    Win32ErrorCodes.ERROR_IPSEC_IKE_NO_POLICY:
        Win32ErrorCodeDescription := 'No policy configured.';
    Win32ErrorCodes.ERROR_IPSEC_IKE_INVALID_SIGNATURE:
        Win32ErrorCodeDescription := 'Failed to verify signature.';
    Win32ErrorCodes.ERROR_IPSEC_IKE_KERBEROS_ERROR:
        Win32ErrorCodeDescription := 'Failed to authenticate using Kerberos.';
    Win32ErrorCodes.ERROR_IPSEC_IKE_NO_PUBLIC_KEY:
        Win32ErrorCodeDescription := 'Peers certificate did not have a public key.';
    Win32ErrorCodes.ERROR_IPSEC_IKE_PROCESS_ERR:
        Win32ErrorCodeDescription := 'Error processing error payload.';
    Win32ErrorCodes.ERROR_IPSEC_IKE_PROCESS_ERR_SA:
        Win32ErrorCodeDescription := 'Error processing SA payload.';
    Win32ErrorCodes.ERROR_IPSEC_IKE_PROCESS_ERR_PROP:
        Win32ErrorCodeDescription := 'Error processing Proposal payload.';
    Win32ErrorCodes.ERROR_IPSEC_IKE_PROCESS_ERR_TRANS:
        Win32ErrorCodeDescription := 'Error processing Transform payload.';
    Win32ErrorCodes.ERROR_IPSEC_IKE_PROCESS_ERR_KE:
        Win32ErrorCodeDescription := 'Error processing KE payload.';
    Win32ErrorCodes.ERROR_IPSEC_IKE_PROCESS_ERR_ID:
        Win32ErrorCodeDescription := 'Error processing ID payload.';
    Win32ErrorCodes.ERROR_IPSEC_IKE_PROCESS_ERR_CERT:
        Win32ErrorCodeDescription := 'Error processing Cert payload.';
    Win32ErrorCodes.ERROR_IPSEC_IKE_PROCESS_ERR_CERT_REQ:
        Win32ErrorCodeDescription := 'Error processing Certificate Request payload.';
    Win32ErrorCodes.ERROR_IPSEC_IKE_PROCESS_ERR_HASH:
        Win32ErrorCodeDescription := 'Error processing Hash payload.';
    Win32ErrorCodes.ERROR_IPSEC_IKE_PROCESS_ERR_SIG:
        Win32ErrorCodeDescription := 'Error processing Signature payload.';
    Win32ErrorCodes.ERROR_IPSEC_IKE_PROCESS_ERR_NONCE:
        Win32ErrorCodeDescription := 'Error processing Nonce payload.';
    Win32ErrorCodes.ERROR_IPSEC_IKE_PROCESS_ERR_NOTIFY:
        Win32ErrorCodeDescription := 'Error processing Notify payload.';
    Win32ErrorCodes.ERROR_IPSEC_IKE_PROCESS_ERR_DELETE:
        Win32ErrorCodeDescription := 'Error processing Delete Payload.';
    Win32ErrorCodes.ERROR_IPSEC_IKE_PROCESS_ERR_VENDOR:
        Win32ErrorCodeDescription := 'Error processing VendorId payload.';
    Win32ErrorCodes.ERROR_IPSEC_IKE_INVALID_PAYLOAD:
        Win32ErrorCodeDescription := 'Invalid payload received.';
    Win32ErrorCodes.ERROR_IPSEC_IKE_LOAD_SOFT_SA:
        Win32ErrorCodeDescription := 'Soft SA loaded.';
    Win32ErrorCodes.ERROR_IPSEC_IKE_SOFT_SA_TORN_DOWN:
        Win32ErrorCodeDescription := 'Soft SA torn down.';
    Win32ErrorCodes.ERROR_IPSEC_IKE_INVALID_COOKIE:
        Win32ErrorCodeDescription := 'Invalid cookie received..';
    Win32ErrorCodes.ERROR_IPSEC_IKE_NO_PEER_CERT:
        Win32ErrorCodeDescription := 'Peer failed to send valid machine certificate.';
    Win32ErrorCodes.ERROR_IPSEC_IKE_PEER_CRL_FAILED:
        Win32ErrorCodeDescription := 'Certification Revocation check of peers certificate failed.';
    Win32ErrorCodes.ERROR_IPSEC_IKE_POLICY_CHANGE:
        Win32ErrorCodeDescription := 'New policy invalidated SAs formed with old policy.';
    Win32ErrorCodes.ERROR_IPSEC_IKE_NO_MM_POLICY:
        Win32ErrorCodeDescription := 'There is no available Main Mode IKE policy.';
    Win32ErrorCodes.ERROR_IPSEC_IKE_NOTCBPRIV:
        Win32ErrorCodeDescription := 'Failed to enabled TCB privilege.';
    Win32ErrorCodes.ERROR_IPSEC_IKE_SECLOADFAIL:
        Win32ErrorCodeDescription := 'Failed to load SECURITY.DLL.';
    Win32ErrorCodes.ERROR_IPSEC_IKE_FAILSSPINIT:
        Win32ErrorCodeDescription :=
            'Failed to obtain security function table dispatch address from SSPI.';
    Win32ErrorCodes.ERROR_IPSEC_IKE_FAILQUERYSSP:
        Win32ErrorCodeDescription := 'Failed to query Kerberos package to obtain max token size.';
    Win32ErrorCodes.ERROR_IPSEC_IKE_SRVACQFAIL:
        Win32ErrorCodeDescription := 'Failed to obtain Kerberos server credentials for ISAKMP/ERROR_IPSEC_IKE service. Kerberos authentication will not function. The most likely reason for this is lack of domain membership. This is normal if your computer is a member of a workgroup.';
    Win32ErrorCodes.ERROR_IPSEC_IKE_SRVQUERYCRED:
        Win32ErrorCodeDescription := 'Failed to determine SSPI principal name for ISAKMP/ERROR_IPSEC_IKE service (QueryCredentialsAttributes).';
    Win32ErrorCodes.ERROR_IPSEC_IKE_GETSPIFAIL:
        Win32ErrorCodeDescription := 'Failed to obtain new SPI for the inbound SA from Ipsec driver. The most common cause for this is that the driver does not have the correct filter. Check your policy to verify the filters.';
    Win32ErrorCodes.ERROR_IPSEC_IKE_INVALID_FILTER:
        Win32ErrorCodeDescription := 'Given filter is invalid.';
    Win32ErrorCodes.ERROR_IPSEC_IKE_OUT_OF_MEMORY:
        Win32ErrorCodeDescription := 'Memory allocation failed.';
    Win32ErrorCodes.ERROR_IPSEC_IKE_ADD_UPDATE_KEY_FAILED:
        Win32ErrorCodeDescription := 'Failed to add Security Association to IPSec Driver. The most common cause for this is if the IKE negotiation took too long to complete. If the problem persists, reduce the load on the faulting machine.';
    Win32ErrorCodes.ERROR_IPSEC_IKE_INVALID_POLICY:
        Win32ErrorCodeDescription := 'Invalid policy.';
    Win32ErrorCodes.ERROR_IPSEC_IKE_UNKNOWN_DOI:
        Win32ErrorCodeDescription := 'Invalid DOI.';
    Win32ErrorCodes.ERROR_IPSEC_IKE_INVALID_SITUATION:
        Win32ErrorCodeDescription := 'Invalid situation.';
    Win32ErrorCodes.ERROR_IPSEC_IKE_DH_FAILURE:
        Win32ErrorCodeDescription := 'Diffie-Hellman failure.';
    Win32ErrorCodes.ERROR_IPSEC_IKE_INVALID_GROUP:
        Win32ErrorCodeDescription := 'Invalid Diffie-Hellman group.';
    Win32ErrorCodes.ERROR_IPSEC_IKE_ENCRYPT:
        Win32ErrorCodeDescription := 'Error encrypting payload.';
    Win32ErrorCodes.ERROR_IPSEC_IKE_DECRYPT:
        Win32ErrorCodeDescription := 'Error decrypting payload.';
    Win32ErrorCodes.ERROR_IPSEC_IKE_POLICY_MATCH:
        Win32ErrorCodeDescription := 'Policy match error.';
    Win32ErrorCodes.ERROR_IPSEC_IKE_UNSUPPORTED_ID:
        Win32ErrorCodeDescription := 'Unsupported ID.';
    Win32ErrorCodes.ERROR_IPSEC_IKE_INVALID_HASH:
        Win32ErrorCodeDescription := 'Hash verification failed.';
    Win32ErrorCodes.ERROR_IPSEC_IKE_INVALID_HASH_ALG:
        Win32ErrorCodeDescription := 'Invalid hash algorithm.';
    Win32ErrorCodes.ERROR_IPSEC_IKE_INVALID_HASH_SIZE:
        Win32ErrorCodeDescription := 'Invalid hash size.';
    Win32ErrorCodes.ERROR_IPSEC_IKE_INVALID_ENCRYPT_ALG:
        Win32ErrorCodeDescription := 'Invalid encryption algorithm.';
    Win32ErrorCodes.ERROR_IPSEC_IKE_INVALID_AUTH_ALG:
        Win32ErrorCodeDescription := 'Invalid authentication algorithm.';
    Win32ErrorCodes.ERROR_IPSEC_IKE_INVALID_SIG:
        Win32ErrorCodeDescription := 'Invalid certificate signature.';
    Win32ErrorCodes.ERROR_IPSEC_IKE_LOAD_FAILED:
        Win32ErrorCodeDescription := 'Load failed.';
    Win32ErrorCodes.ERROR_IPSEC_IKE_RPC_DELETE:
        Win32ErrorCodeDescription := 'Deleted via RPC call.';
    Win32ErrorCodes.ERROR_IPSEC_IKE_BENIGN_REINIT:
        Win32ErrorCodeDescription :=
            'Temporary state created to perform reinitialization. This is not a real failure.';
    Win32ErrorCodes.ERROR_IPSEC_IKE_INVALID_RESPONDER_LIFETIME_NOTIFY:
        Win32ErrorCodeDescription := 'The lifetime value received in the Responder Lifetime Notify is below the Windows 2000 configured minimum value. Please fix the policy on the peer machine.';
    Win32ErrorCodes.ERROR_IPSEC_IKE_QM_LIMIT_REAP:
        Win32ErrorCodeDescription := 'SA reaped because QM limit was reached.';
    Win32ErrorCodes.ERROR_IPSEC_IKE_INVALID_CERT_KEYLEN:
        Win32ErrorCodeDescription :=
            'Key length in certificate is too small for configured security requirements.';
    Win32ErrorCodes.ERROR_IPSEC_IKE_MM_LIMIT:
        Win32ErrorCodeDescription := 'Max number of established MM SAs to peer exceeded.';
    Win32ErrorCodes.ERROR_IPSEC_IKE_NEGOTIATION_DISABLED:
        Win32ErrorCodeDescription := 'IKE received a policy that disables negotiation.';
    Win32ErrorCodes.ERROR_IPSEC_IKE_QM_LIMIT:
        Win32ErrorCodeDescription :=
            'Reached maximum quick mode limit for the main mode. New main mode will be started.';
ELSE
    Win32ErrorCodeDescription := 'Unknown Win32 error code.';
END_CASE

END_FUNCTION

// ---- NC_Tests/ToNcErrorCode_Tests.TcPOU
FUNCTION_BLOCK ToNcErrorCode_Tests EXTENDS FB_TestSuite

ConversionOfValidErrorCode();
ConversionOfInvalidErrorCode();

METHOD ConversionOfInvalidErrorCode
TcUnit.TEST('ConversionOfInvalidErrorCode');

AssertEquals_DINT(
    Expected:=NcErrorCodes.ERR_UNKNOWN,
    Actual:=ToNcErrorCode(1234567),
    Message:='Error conversion not correct.'
);

TcUnit.TEST_FINISHED();
END_METHOD

METHOD ConversionOfValidErrorCode
TcUnit.TEST('ConversionOfValidErrorCode');

AssertEquals_UDINT(
    Expected:=NcErrorCodes.CONTROLLER_ERROR_DRIVE_ADDRESS,
    Actual:=ToNcErrorCode(17730),
    Message:='Error conversion not correct.'
);

TcUnit.TEST_FINISHED();
END_METHOD

END_FUNCTION_BLOCK

// ---- NC/ToNcErrorCode.TcPOU
(*
Convert a NC error code of type UDINT to the NcErrorCodes datatype.

## Example
```
ncErrorId := 17693;
ncErrorCode := ToNcErrorCode(ncErrorId); // CONTROLLER_ERROR_DEAD_RANGE_NOT_ALLOWED;
```

## Source
https://infosys.beckhoff.com/content/1033/tc3ncerrcode/1521556875.html?id=2911757239699425890
*)
FUNCTION ToNcErrorCode : NcErrorCodes
VAR_INPUT
    errorCode : UDINT;
END_VAR

CASE errorCode OF
    17664:
        ToNcErrorCode := NcErrorCodes.CONTROLLER_ERROR_CONTROLLER_ID_NOT_ALLOWED;
    17665:
        ToNcErrorCode := NcErrorCodes.CONTROLLER_ERROR_CONTROLLER_TYPE_NOT_ALLOWED;
    17666:
        ToNcErrorCode := NcErrorCodes.CONTROLLER_ERROR_OPERATION_MODE_CONTROLLER_NOT_ALLOWED;
    17667:
        ToNcErrorCode :=
            NcErrorCodes.CONTROLLER_ERROR_WEIGHTING_OF_THE_VELOCITY_PRE_CONTROL_NOT_ALLOWED;
    17668:
        ToNcErrorCode := NcErrorCodes.CONTROLLER_ERROR_LAG_ERROR_MONITOR_POSITION_NOT_ALLOWED;
    17669:
        ToNcErrorCode := NcErrorCodes.CONTROLLER_ERROR_LAG_MONITORING_VELOCITY_NOT_ALLOWED;
    17670:
        ToNcErrorCode := NcErrorCodes.CONTROLLER_ERROR_LAG_ERROR_WINDOW_POSITION_NOT_ALLOWED;
    17671:
        ToNcErrorCode := NcErrorCodes.CONTROLLER_ERROR_LAG_ERROR_FILTER_TIME_POSITION_NOT_ALLOWED;
    17672:
        ToNcErrorCode := NcErrorCodes.CONTROLLER_ERROR_LAG_ERROR_WINDOW_VELOCITY_NOT_ALLOWED;
    17673:
        ToNcErrorCode := NcErrorCodes.CONTROLLER_ERROR_LAG_ERROR_FILTER_TIME_VELOCITY_NOT_ALLOWED;
    17674:
        ToNcErrorCode := NcErrorCodes
            .CONTROLLER_ERROR_CONTROLLER_OUTPUT_LIMITATION_OUTPUT_LIMITATION_NOT_ALLOWED;
    17680:
        ToNcErrorCode :=
            NcErrorCodes.CONTROLLER_ERROR_PROPORTIONAL_GAIN_KV_OR_KP_CONTROLLER_NOT_ALLOWED;
    17681:
        ToNcErrorCode :=
            NcErrorCodes.CONTROLLER_ERROR_INTEGRAL_ACTION_TIME_TN_CONTROLLER_NOT_ALLOWED_POSITION;
    17682:
        ToNcErrorCode :=
            NcErrorCodes.CONTROLLER_ERROR_RATE_TIME_TV_CONTROLLER_NOT_ALLOWED_POSITION;
    17683:
        ToNcErrorCode :=
            NcErrorCodes.CONTROLLER_ERROR_DAMPING_TIME_TD_CONTROLLER_NOT_ALLOWED_POSITION;
    17684:
        ToNcErrorCode := NcErrorCodes
            .CONTROLLER_ERROR_ACTIVATION_OF_THE_AUTOMATIC_OFFSET_CALIBRATION_NOT_ALLOWED;
    17685:
        ToNcErrorCode := NcErrorCodes
            .CONTROLLER_ERROR_ADDITIONAL_PROPORTIONAL_GAIN_KV_OR_KP_CONTROLLER_NOT_ALLOWED;
    17686:
        ToNcErrorCode := NcErrorCodes
            .CONTROLLER_ERROR_REFERENCE_VELOCITY_FOR_ADDITIONAL_PROP_GAIN_CONTROLLER_NOT_ALLOWED;
    17687:
        ToNcErrorCode := NcErrorCodes.CONTROLLER_ERROR_PROPORTIONAL_GAIN_PA_PROPORTION_NOT_ALLOWED;
    17688:
        ToNcErrorCode := NcErrorCodes.CONTROLLER_ERROR_PROPORTIONAL_GAIN_KV_CONTROLLER_NOT_ALLOWED;
    17689:
        ToNcErrorCode :=
            NcErrorCodes.CONTROLLER_ERROR_INTEGRAL_ACTION_TIME_TN_CONTROLLER_NOT_ALLOWED_VELOCITY;
    17692:
        ToNcErrorCode := NcErrorCodes.CONTROLLER_ERROR_VELOCITY_FILTER_TIME_NOT_ALLOWED;
    17693:
        ToNcErrorCode := NcErrorCodes.CONTROLLER_ERROR_DEAD_RANGE_NOT_ALLOWED;
    17695:
        ToNcErrorCode := NcErrorCodes.CONTROLLER_ERROR_PROPORTIONAL_GAIN_KCP_NOT_ALLOWED;
    17696:
        ToNcErrorCode := NcErrorCodes.CONTROLLER_ERROR_RATE_TIME_TV_CONTROLLER_NOT_ALLOWED;
    17697:
        ToNcErrorCode := NcErrorCodes.CONTROLLER_ERROR_DAMPING_TIME_TD_CONTROLLER_NOT_ALLOWED;
    17698:
        ToNcErrorCode := NcErrorCodes.CONTROLLER_ERROR_LIMITATION_OF_THE_I_PART_NOT_ALLOWED;
    17699:
        ToNcErrorCode := NcErrorCodes.CONTROLLER_ERROR_LIMITATION_OF_THE_D_PART_NOT_ALLOWED;
    17700:
        ToNcErrorCode := NcErrorCodes
            .CONTROLLER_ERROR_PARAMETER_DEACTIVATION_OF_THE_I_PART_DURING_TRAVEL_NOT_ALLOWED;
    17701:
        ToNcErrorCode :=
            NcErrorCodes.CONTROLLER_ERROR_PARAMETER_FILTER_TIME_FOR_P_T2_FILTER_NOT_ALLOWED;
    17702:
        ToNcErrorCode :=
            NcErrorCodes.CONTROLLER_ERROR_VELOCITY_OBSERVER_PARAMETERIZED_MODE_IS_NOT_ALLOWED;
    17703:
        ToNcErrorCode := NcErrorCodes
            .CONTROLLER_ERROR_VELOCITY_OBSERVER_MOTOR_TORQUE_CONSTANT_KT_OR_KF_IS_NOT_ALLOWED;
    17704:
        ToNcErrorCode := NcErrorCodes
            .CONTROLLER_ERROR_VELOCITY_OBSERVER_MOTOR_MOMENT_OF_INERTIA_JM_IS_NOT_ALLOWED;
    17705:
        ToNcErrorCode :=
            NcErrorCodes.CONTROLLER_ERROR_VELOCITY_OBSERVER_BANDWIDTH_F0_IS_NOT_ALLOWED;
    17706:
        ToNcErrorCode :=
            NcErrorCodes.CONTROLLER_ERROR_VELOCITY_OBSERVER_CORRECTION_FACTOR_KC_IS_NOT_ALLOWED;
    17707:
        ToNcErrorCode := NcErrorCodes
            .CONTROLLER_ERROR_VELOCITY_OBSERVER_TIME_CONSTANT_T_FOR_1ST_ORDER_FILTER_NOT_ALLOWED;
    17708:
        ToNcErrorCode := NcErrorCodes
            .CONTROLLER_ERROR_VELOCITY_OBSERVER_AMPLITUDE_DAMPING_FOR_2ND_ORDER_FILTER_NOT_ALLOWED;
    17709:
        ToNcErrorCode := NcErrorCodes
            .CONTROLLER_ERROR_VELOCITY_OBSERVER_FREQUENCY_FOR_2ND_ORDER_FILTER_NOT_ALLOWED;
    17728:
        ToNcErrorCode := NcErrorCodes.CONTROLLER_ERROR_CONTROLLER_INITIALIZATION;
    17729:
        ToNcErrorCode := NcErrorCodes.CONTROLLER_ERROR_AXIS_ADDRESS;
    17730:
        ToNcErrorCode := NcErrorCodes.CONTROLLER_ERROR_DRIVE_ADDRESS;
    17744:
        ToNcErrorCode := NcErrorCodes.CONTROLLER_ERROR_LAG_ERROR_MONITOR_POSITION;
    17745:
        ToNcErrorCode := NcErrorCodes.CONTROLLER_ERROR_LAG_MONITORING_VELOCITY;
    17824:
        ToNcErrorCode := NcErrorCodes.CONTROLLER_ERROR_INTERNAL_ERROR_CONTROLERR_RANGE_AREA_ASIDE;
    17825:
        ToNcErrorCode := NcErrorCodes.CONTROLLER_ERROR_INTERNAL_ERROR_CONTROLERR_RANGE_AREA_BSIDE;
    17826:
        ToNcErrorCode := NcErrorCodes.CONTROLLER_ERROR_INTERNAL_ERROR_CONTROLERR_RANGE_QNENN;
    17827:
        ToNcErrorCode := NcErrorCodes.CONTROLLER_ERROR_INTERNAL_ERROR_CONTROLERR_RANGE_PNENN;
    17828:
        ToNcErrorCode :=
            NcErrorCodes.CONTROLLER_ERROR_INTERNAL_ERROR_CONTROLERR_RANGE_AXISIDPRESP0;
ELSE
    ToNcErrorCode := NcErrorCodes.ERR_UNKNOWN;
END_CASE

END_FUNCTION

// ---- NC_Tests/NcErrorCodeDesciption_Tests.TcPOU
{attribute 'hide'}
FUNCTION_BLOCK NcErrorCodeDesciption_Tests EXTENDS TcUnit.FB_TestSuite

DescriptionOfKnownErrorCode();
DescriptionOfUnknownErrorCode();

METHOD DescriptionOfKnownErrorCode
TcUnit.TEST('DescriptionOfKnownErrorCode');

AssertEquals_STRING(
    Expected:='The controller has not been initialized. Although the controller has been created, the rest of the initialization has not been performed (1. Initialization of controller, 2. Reset of controller).',
    Actual:=NcErrorCodeDescription(NcErrorCodes.CONTROLLER_ERROR_CONTROLLER_INITIALIZATION),
    Message:='Error description not correct.'
);

TcUnit.TEST_FINISHED();
END_METHOD

METHOD DescriptionOfUnknownErrorCode
TcUnit.TEST('DescriptionOfUnknownErrorCode');

AssertEquals_STRING(
    Expected:='Unknown NC error code.',
    Actual:=NcErrorCodeDescription(NcErrorCodes.ERR_UNKNOWN),
    Message:='Error description not correct.'
);

TcUnit.TEST_FINISHED();
END_METHOD

END_FUNCTION_BLOCK

// ---- NC/NcErrorCodeDescription.TcPOU
(*
Returns an description of the error from the NcErrorCodes datatype.

## Example
```
ncErrorCode := NcErrorCodes.CONTROLLER_ERROR_LAG_ERROR_WINDOW_VELOCITY_NOT_ALLOWED;
errorDescription := NcErrorCodeDescription(ncErrorCode); // 'The value for the lag error window (velocity) is not allowed.'
```

## Source
https://infosys.beckhoff.com/content/1033/tc3ncerrcode/1521556875.html?id=2911757239699425890
*)
FUNCTION NcErrorCodeDescription : T_MaxString
VAR_INPUT
    ncErrorCode : NcErrorCodes;
END_VAR

CASE ncErrorCode OF
    NcErrorCodes.CONTROLLER_ERROR_CONTROLLER_ID_NOT_ALLOWED:
        NcErrorCodeDescription := 'The value for the controller ID is not allowed, e.g. because it has already been assigned, is less than or equal to zero, or is greater than 255.';
    NcErrorCodes.CONTROLLER_ERROR_CONTROLLER_TYPE_NOT_ALLOWED:
        NcErrorCodeDescription :=
            'The value for the controller type is unacceptable because it is not defined.';
    NcErrorCodes.CONTROLLER_ERROR_OPERATION_MODE_CONTROLLER_NOT_ALLOWED:
        NcErrorCodeDescription := 'The value for the controller operating mode is not allowed.';
    NcErrorCodes.CONTROLLER_ERROR_WEIGHTING_OF_THE_VELOCITY_PRE_CONTROL_NOT_ALLOWED:
        NcErrorCodeDescription :=
            'The value for the percentage weighting of the velocity pre-control is not allowed.';
    NcErrorCodes.CONTROLLER_ERROR_LAG_ERROR_MONITOR_POSITION_NOT_ALLOWED:
        NcErrorCodeDescription :=
            'The value for the activation of the lag error monitor is not allowed.';
    NcErrorCodes.CONTROLLER_ERROR_LAG_MONITORING_VELOCITY_NOT_ALLOWED:
        NcErrorCodeDescription :=
            'The value for the activation of the lag error monitoring (velocity) is not allowed.';
    NcErrorCodes.CONTROLLER_ERROR_LAG_ERROR_WINDOW_POSITION_NOT_ALLOWED:
        NcErrorCodeDescription :=
            'The value for the lag error window (maximum allowable lag error) is not allowed.';
    NcErrorCodes.CONTROLLER_ERROR_LAG_ERROR_FILTER_TIME_POSITION_NOT_ALLOWED:
        NcErrorCodeDescription :=
            'The value for the lag error filter time (position) is not allowed.';
    NcErrorCodes.CONTROLLER_ERROR_LAG_ERROR_WINDOW_VELOCITY_NOT_ALLOWED:
        NcErrorCodeDescription := 'The value for the lag error window (velocity) is not allowed.';
    NcErrorCodes.CONTROLLER_ERROR_LAG_ERROR_FILTER_TIME_VELOCITY_NOT_ALLOWED:
        NcErrorCodeDescription :=
            'The value for the lag error filter time (velocity) is not allowed.';
    NcErrorCodes.CONTROLLER_ERROR_CONTROLLER_OUTPUT_LIMITATION_OUTPUT_LIMITATION_NOT_ALLOWED:
        NcErrorCodeDescription := 'The value for the output limitation of the controller at the total manipulated variable is invalid.';
    NcErrorCodes.CONTROLLER_ERROR_PROPORTIONAL_GAIN_KV_OR_KP_CONTROLLER_NOT_ALLOWED:
        NcErrorCodeDescription :=
            'The value for the proportional gain (Kv factor or Kp factor) is not allowed.';
    NcErrorCodes.CONTROLLER_ERROR_INTEGRAL_ACTION_TIME_TN_CONTROLLER_NOT_ALLOWED_POSITION:
        NcErrorCodeDescription :=
            'The value for the integral action time is not allowed (I part of the PID T1 controller).';
    NcErrorCodes.CONTROLLER_ERROR_RATE_TIME_TV_CONTROLLER_NOT_ALLOWED_POSITION:
        NcErrorCodeDescription := 'The value for the derivative action time is not allowed (D part of the PID T1 controller).';
    NcErrorCodes.CONTROLLER_ERROR_DAMPING_TIME_TD_CONTROLLER_NOT_ALLOWED_POSITION:
        NcErrorCodeDescription :=
            'The value for the damping time is not allowed (D part of the PID T1 controller).';
    NcErrorCodes.CONTROLLER_ERROR_ACTIVATION_OF_THE_AUTOMATIC_OFFSET_CALIBRATION_NOT_ALLOWED:
        NcErrorCodeDescription := 'Activation of the automatic offset calibration is only possible for certain types of controller (with no I component).';
    NcErrorCodes.CONTROLLER_ERROR_ADDITIONAL_PROPORTIONAL_GAIN_KV_OR_KP_CONTROLLER_NOT_ALLOWED:
        NcErrorCodeDescription := 'The value for the second term of the proportional gain (Kv factor or Kp factor) is not allowed.';
    NcErrorCodes
        .CONTROLLER_ERROR_REFERENCE_VELOCITY_FOR_ADDITIONAL_PROP_GAIN_CONTROLLER_NOT_ALLOWED:
        NcErrorCodeDescription := 'The value for the reference velocity percentage data entry, to which the additional proportional gain is applied, is not allowed.';
    NcErrorCodes.CONTROLLER_ERROR_PROPORTIONAL_GAIN_PA_PROPORTION_NOT_ALLOWED:
        NcErrorCodeDescription :=
            'The value for the proportional gain (Pa factor) is not allowed.';
    NcErrorCodes.CONTROLLER_ERROR_PROPORTIONAL_GAIN_KV_CONTROLLER_NOT_ALLOWED:
        NcErrorCodeDescription :=
            'The value for the proportional gain (Kv factor) is not allowed.';
    NcErrorCodes.CONTROLLER_ERROR_INTEGRAL_ACTION_TIME_TN_CONTROLLER_NOT_ALLOWED_VELOCITY:
        NcErrorCodeDescription :=
            'The value for the integral action time is not allowed (I part of the PID T1 controller).';
    NcErrorCodes.CONTROLLER_ERROR_VELOCITY_FILTER_TIME_NOT_ALLOWED:
        NcErrorCodeDescription :=
            'The parameter for the velocity filter time in seconds is invalid (P-T1 filter).';
    NcErrorCodes.CONTROLLER_ERROR_DEAD_RANGE_NOT_ALLOWED:
        NcErrorCodeDescription := 'The value for the dead range (neutral zone) of the position error or the velocity error (control deviation) is not allowed.';
    NcErrorCodes.CONTROLLER_ERROR_PROPORTIONAL_GAIN_KCP_NOT_ALLOWED:
        NcErrorCodeDescription := 'The parameter for the proportional gain Kcp of the slave coupling difference control is invalid.';
    NcErrorCodes.CONTROLLER_ERROR_RATE_TIME_TV_CONTROLLER_NOT_ALLOWED:
        NcErrorCodeDescription := 'The value for the derivative action time is not allowed (D part of the PID T1 controller).';
    NcErrorCodes.CONTROLLER_ERROR_DAMPING_TIME_TD_CONTROLLER_NOT_ALLOWED:
        NcErrorCodeDescription :=
            'The value for the damping time is not allowed (D part of the PID T1 controller).';
    NcErrorCodes.CONTROLLER_ERROR_LIMITATION_OF_THE_I_PART_NOT_ALLOWED:
        NcErrorCodeDescription :=
            'The parameter for limiting the I-part of a PI- or PID-controller is not allowed.';
    NcErrorCodes.CONTROLLER_ERROR_LIMITATION_OF_THE_D_PART_NOT_ALLOWED:
        NcErrorCodeDescription :=
            'The parameter for limiting the D-part of a PI- or PID-controller is not allowed.';
    NcErrorCodes.CONTROLLER_ERROR_PARAMETER_DEACTIVATION_OF_THE_I_PART_DURING_TRAVEL_NOT_ALLOWED:
        NcErrorCodeDescription :=
            'The boolean parameter for switching off the I-part during active positioning is invalid.';
    NcErrorCodes.CONTROLLER_ERROR_PARAMETER_FILTER_TIME_FOR_P_T2_FILTER_NOT_ALLOWED:
        NcErrorCodeDescription := 'The time T0 in seconds is not permissible as a filter time for the P-T2 element of the velocity controller.';
    NcErrorCodes.CONTROLLER_ERROR_VELOCITY_OBSERVER_PARAMETERIZED_MODE_IS_NOT_ALLOWED:
        NcErrorCodeDescription := 'The parameterized mode (0=OFF, 1=LUENBERGER) for the velocity observer of the special NC controller in the torque interface is not permitted.';
    NcErrorCodes.CONTROLLER_ERROR_VELOCITY_OBSERVER_MOTOR_TORQUE_CONSTANT_KT_OR_KF_IS_NOT_ALLOWED:
        NcErrorCodeDescription := 'The parameter for the motor torque constant Kt (rotary motor) or Kf (linear motor) of the velocity observer of the special NC controller in the torque interface is invalid.';
    NcErrorCodes.CONTROLLER_ERROR_VELOCITY_OBSERVER_MOTOR_MOMENT_OF_INERTIA_JM_IS_NOT_ALLOWED:
        NcErrorCodeDescription := 'The parameter for the motor moment of inertia JM of the velocity observer of the special NC controller in the torque interface is invalid.';
    NcErrorCodes.CONTROLLER_ERROR_VELOCITY_OBSERVER_BANDWIDTH_F0_IS_NOT_ALLOWED:
        NcErrorCodeDescription := 'The parameter for the bandwidth f0 of the velocity observer of the special NC controller in the torque interface is invalid.';
    NcErrorCodes.CONTROLLER_ERROR_VELOCITY_OBSERVER_CORRECTION_FACTOR_KC_IS_NOT_ALLOWED:
        NcErrorCodeDescription := 'The parameter for the correction factor kc of the velocity observer of the special NC controller in the torque interface is invalid.';
    NcErrorCodes
        .CONTROLLER_ERROR_VELOCITY_OBSERVER_TIME_CONSTANT_T_FOR_1ST_ORDER_FILTER_NOT_ALLOWED:
        NcErrorCodeDescription := 'The time constant T for the 1st order velocity filter (PID-T2 or "Lead Lag") of the velocity observer of the special NC controller in the torque interface is not allowed.';
    NcErrorCodes
        .CONTROLLER_ERROR_VELOCITY_OBSERVER_AMPLITUDE_DAMPING_FOR_2ND_ORDER_FILTER_NOT_ALLOWED:
        NcErrorCodeDescription := 'The high-pass/low-pass amplitude attenuation dHP or dTP for the 2nd order velocity filter ("bi-quad") of the velocity observer of the special NC controller in the torque interface is not allowed.';
    NcErrorCodes.CONTROLLER_ERROR_VELOCITY_OBSERVER_FREQUENCY_FOR_2ND_ORDER_FILTER_NOT_ALLOWED:
        NcErrorCodeDescription := 'The high-pass/low-pass frequency fHP or fTP for the 2nd order velocity filter ("bi-quad") of the velocity observer of the special NC controller in the torque interface is not allowed.';
    NcErrorCodes.CONTROLLER_ERROR_CONTROLLER_INITIALIZATION:
        NcErrorCodeDescription := 'The controller has not been initialized. Although the controller has been created, the rest of the initialization has not been performed (1. Initialization of controller, 2. Reset of controller).';
    NcErrorCodes.CONTROLLER_ERROR_AXIS_ADDRESS:
        NcErrorCodeDescription :=
            'The controller does not know its axis, or the axis address has not been initialized.';
    NcErrorCodes.CONTROLLER_ERROR_DRIVE_ADDRESS:
        NcErrorCodeDescription :=
            'The controller does not know its drive, or the drive address has not been initialized.';
    NcErrorCodes.CONTROLLER_ERROR_LAG_ERROR_MONITOR_POSITION:
        NcErrorCodeDescription := 'While the lag error monitor was active (position), the lag error was exceeded by an amount greater than the lag error window and which lasting longer than the parameterized lag error filter time.';
    NcErrorCodes.CONTROLLER_ERROR_LAG_MONITORING_VELOCITY:
        NcErrorCodeDescription := 'With active lag error monitoring (velocity) a velocity lag error exceedance has occurred, whose magnitude is greater than the lag error window, and whose duration is longer than the parameterized lag error filter time.';
    NcErrorCodes.CONTROLLER_ERROR_INTERNAL_ERROR_CONTROLERR_RANGE_AREA_ASIDE:
        NcErrorCodeDescription := 'Internal error: CONTROLERR_RANGE_AREA_ASIDE';
    NcErrorCodes.CONTROLLER_ERROR_INTERNAL_ERROR_CONTROLERR_RANGE_AREA_BSIDE:
        NcErrorCodeDescription := 'Internal error: CONTROLERR_RANGE_AREA_BSIDE';
    NcErrorCodes.CONTROLLER_ERROR_INTERNAL_ERROR_CONTROLERR_RANGE_QNENN:
        NcErrorCodeDescription := 'Internal error: CONTROLERR_RANGE_QNENN';
    NcErrorCodes.CONTROLLER_ERROR_INTERNAL_ERROR_CONTROLERR_RANGE_PNENN:
        NcErrorCodeDescription := 'Internal error: CONTROLERR_RANGE_PNENN';
    NcErrorCodes.CONTROLLER_ERROR_INTERNAL_ERROR_CONTROLERR_RANGE_AXISIDPRESP0:
        NcErrorCodeDescription := 'Internal error: CONTROLERR_RANGE_AXISIDPRESP0';
    NcErrorCodes.ERR_UNKNOWN:
        NcErrorCodeDescription := 'Unknown NC error code.';
ELSE
    NcErrorCodeDescription := 'Error code not recognized';
END_CASE

END_FUNCTION

// ---- ADS/AdsErrorCodeDescription.TcPOU
(*
Returns an description of the error from the AdsErrorCodes datatype.

## Example
```
adsErrorCode := AdsErrorCodes.ADSERR_DEVICE_NOMEMORY;
errorDescription := TcError.AdsErrorCodeDescription(adsErrorCode); // 'Insufficient memory.'
```

## Source
https://infosys.beckhoff.com/content/1033/tf6701_tc3_iot_communication_mqtt/374277003.html?id=1376723717835500292
*)
FUNCTION AdsErrorCodeDescription : T_MaxString
VAR_INPUT
    adsErrorCode : AdsErrorCodes;
END_VAR

CASE adsErrorCode OF
    AdsErrorCodes.ERR_NOERROR:
        AdsErrorCodeDescription := 'No error.';
    AdsErrorCodes.ERR_INTERNAL:
        AdsErrorCodeDescription := 'Internal error.';
    AdsErrorCodes.ERR_NORTIME:
        AdsErrorCodeDescription := 'No real-time.';
    AdsErrorCodes.ERR_ALLOCLOCKEDMEM:
        AdsErrorCodeDescription := 'Allocation locked – memory error.';
    AdsErrorCodes.ERR_INSERTMAILBOX:
        AdsErrorCodeDescription := 'Mailbox full – the ADS message could not be sent. Reducing the number of ADS messages per cycle will help.';
    AdsErrorCodes.ERR_WRONGRECEIVEHMSG:
        AdsErrorCodeDescription := 'Wrong HMSG.';
    AdsErrorCodes.ERR_TARGETPORTNOTFOUND:
        AdsErrorCodeDescription :=
            'Target port not found – ADS server is not started or is not reachable.';
    AdsErrorCodes.ERR_TARGETMACHINENOTFOUND:
        AdsErrorCodeDescription := 'Target computer not found – AMS route was not found.';
    AdsErrorCodes.ERR_UNKNOWNCMDID:
        AdsErrorCodeDescription := 'Unknown command ID.';
    AdsErrorCodes.ERR_BADTASKID:
        AdsErrorCodeDescription := 'Invalid task ID.';
    AdsErrorCodes.ERR_NOIO:
        AdsErrorCodeDescription := 'No IO.';
    AdsErrorCodes.ERR_UNKNOWNAMSCMD:
        AdsErrorCodeDescription := 'Unknown AMS command.';
    AdsErrorCodes.ERR_WIN32ERROR:
        AdsErrorCodeDescription := 'Win32 error.';
    AdsErrorCodes.ERR_PORTNOTCONNECTED:
        AdsErrorCodeDescription := 'Port not connected.';
    AdsErrorCodes.ERR_INVALIDAMSLENGTH:
        AdsErrorCodeDescription := 'Invalid AMS length.';
    AdsErrorCodes.ERR_INVALIDAMSNETID:
        AdsErrorCodeDescription := 'Invalid AMS Net ID.';
    AdsErrorCodes.ERR_LOWINSTLEVEL:
        AdsErrorCodeDescription := 'Installation level is too low –TwinCAT 2 license error.';
    AdsErrorCodes.ERR_NODEBUGINTAVAILABLE:
        AdsErrorCodeDescription := 'No debugging available.';
    AdsErrorCodes.ERR_PORTDISABLED:
        AdsErrorCodeDescription := 'Port disabled – TwinCAT system service not started.';
    AdsErrorCodes.ERR_PORTALREADYCONNECTED:
        AdsErrorCodeDescription := 'Port already connected.';
    AdsErrorCodes.ERR_AMSSYNC_W32ERROR:
        AdsErrorCodeDescription := 'AMS Sync Win32 error.';
    AdsErrorCodes.ERR_AMSSYNC_TIMEOUT:
        AdsErrorCodeDescription := 'AMS Sync Timeout.';
    AdsErrorCodes.ERR_AMSSYNC_AMSERROR:
        AdsErrorCodeDescription := 'AMS Sync error.';
    AdsErrorCodes.ERR_AMSSYNC_NOINDEXINMAP:
        AdsErrorCodeDescription := 'No index map for AMS Sync available.';
    AdsErrorCodes.ERR_INVALIDAMSPORT:
        AdsErrorCodeDescription := 'Invalid AMS port.';
    AdsErrorCodes.ERR_NOMEMORY:
        AdsErrorCodeDescription := 'No memory.';
    AdsErrorCodes.ERR_TCPSEND:
        AdsErrorCodeDescription := 'TCP send error.';
    AdsErrorCodes.ERR_HOSTUNREACHABLE:
        AdsErrorCodeDescription := 'Host unreachable.';
    AdsErrorCodes.ERR_INVALIDAMSFRAGMENT:
        AdsErrorCodeDescription := 'Invalid AMS fragment.';
    AdsErrorCodes.ERR_TLSSEND:
        AdsErrorCodeDescription := 'TLS send error – secure ADS connection failed.';
    AdsErrorCodes.ERR_ACCESSDENIED:
        AdsErrorCodeDescription := 'Access denied – secure ADS access denied.';
    AdsErrorCodes.ROUTERERR_NOLOCKEDMEMORY:
        AdsErrorCodeDescription := 'Locked memory cannot be allocated.';
    AdsErrorCodes.ROUTERERR_RESIZEMEMORY:
        AdsErrorCodeDescription := 'The router memory size could not be changed.';
    AdsErrorCodes.ROUTERERR_MAILBOXFULL:
        AdsErrorCodeDescription :=
            'The mailbox has reached the maximum number of possible messages.';
    AdsErrorCodes.ROUTERERR_DEBUGBOXFULL:
        AdsErrorCodeDescription :=
            'The Debug mailbox has reached the maximum number of possible messages.';
    AdsErrorCodes.ROUTERERR_UNKNOWNPORTTYPE:
        AdsErrorCodeDescription := 'The port type is unknown.';
    AdsErrorCodes.ROUTERERR_NOTINITIALIZED:
        AdsErrorCodeDescription := 'The router is not initialized.';
    AdsErrorCodes.ROUTERERR_PORTALREADYINUSE:
        AdsErrorCodeDescription := 'The port number is already assigned.';
    AdsErrorCodes.ROUTERERR_NOTREGISTERED:
        AdsErrorCodeDescription := 'The port is not registered.';
    AdsErrorCodes.ROUTERERR_NOMOREQUEUES:
        AdsErrorCodeDescription := 'The maximum number of ports has been reached.';
    AdsErrorCodes.ROUTERERR_INVALIDPORT:
        AdsErrorCodeDescription := 'The port is invalid.';
    AdsErrorCodes.ROUTERERR_NOTACTIVATED:
        AdsErrorCodeDescription := 'The router is not active.';
    AdsErrorCodes.ROUTERERR_FRAGMENTBOXFULL:
        AdsErrorCodeDescription :=
            'The mailbox has reached the maximum number for fragmented messages.';
    AdsErrorCodes.ROUTERERR_FRAGMENTTIMEOUT:
        AdsErrorCodeDescription := 'A fragment timeout has occurred.';
    AdsErrorCodes.ROUTERERR_TOBEREMOVED:
        AdsErrorCodeDescription := 'The port is removed.';
    AdsErrorCodes.ADSERR_DEVICE_ERROR:
        AdsErrorCodeDescription := 'General device error.';
    AdsErrorCodes.ADSERR_DEVICE_SRVNOTSUPP:
        AdsErrorCodeDescription := 'Service is not supported by the server.';
    AdsErrorCodes.ADSERR_DEVICE_INVALIDGRP:
        AdsErrorCodeDescription := 'Invalid index group.';
    AdsErrorCodes.ADSERR_DEVICE_INVALIDOFFSET:
        AdsErrorCodeDescription := 'Invalid index offset.';
    AdsErrorCodes.ADSERR_DEVICE_INVALIDACCESS:
        AdsErrorCodeDescription := 'Reading or writing not permitted.';
    AdsErrorCodes.ADSERR_DEVICE_INVALIDSIZE:
        AdsErrorCodeDescription := 'Parameter size not correct.';
    AdsErrorCodes.ADSERR_DEVICE_INVALIDDATA:
        AdsErrorCodeDescription := 'Invalid data values.';
    AdsErrorCodes.ADSERR_DEVICE_NOTREADY:
        AdsErrorCodeDescription := 'Device is not ready to operate.';
    AdsErrorCodes.ADSERR_DEVICE_BUSY:
        AdsErrorCodeDescription := 'Device is busy.';
    AdsErrorCodes.ADSERR_DEVICE_INVALIDCONTEXT:
        AdsErrorCodeDescription := 'Invalid operating system context. This can result from use of ADS function blocks in different tasks. It may be possible to resolve this through Multi-task data access synchronization in the PLC.';
    AdsErrorCodes.ADSERR_DEVICE_NOMEMORY:
        AdsErrorCodeDescription := 'Insufficient memory.';
    AdsErrorCodes.ADSERR_DEVICE_INVALIDPARM:
        AdsErrorCodeDescription := 'Invalid parameter values.';
    AdsErrorCodes.ADSERR_DEVICE_NOTFOUND:
        AdsErrorCodeDescription := 'Not found (files, ...).';
    AdsErrorCodes.ADSERR_DEVICE_SYNTAX:
        AdsErrorCodeDescription := 'Syntax error in file or command.';
    AdsErrorCodes.ADSERR_DEVICE_INCOMPATIBLE:
        AdsErrorCodeDescription := 'Objects do not match.';
    AdsErrorCodes.ADSERR_DEVICE_EXISTS:
        AdsErrorCodeDescription := 'Object already exists.';
    AdsErrorCodes.ADSERR_DEVICE_SYMBOLNOTFOUND:
        AdsErrorCodeDescription := 'Symbol not found.';
    AdsErrorCodes.ADSERR_DEVICE_SYMBOLVERSIONINVALID:
        AdsErrorCodeDescription :=
            'Invalid symbol version. This can occur due to an online change. Create a new handle.';
    AdsErrorCodes.ADSERR_DEVICE_INVALIDSTATE:
        AdsErrorCodeDescription := 'Device (server) is in invalid state.';
    AdsErrorCodes.ADSERR_DEVICE_TRANSMODENOTSUPP:
        AdsErrorCodeDescription := 'AdsTransMode not supported.';
    AdsErrorCodes.ADSERR_DEVICE_NOTIFYHNDINVALID:
        AdsErrorCodeDescription := 'Notification handle is invalid.';
    AdsErrorCodes.ADSERR_DEVICE_CLIENTUNKNOWN:
        AdsErrorCodeDescription := 'Notification client not registered.';
    AdsErrorCodes.ADSERR_DEVICE_NOMOREHDLS:
        AdsErrorCodeDescription := 'No further handle available.';
    AdsErrorCodes.ADSERR_DEVICE_INVALIDWATCHSIZE:
        AdsErrorCodeDescription := 'Notification size too large.';
    AdsErrorCodes.ADSERR_DEVICE_NOTINIT:
        AdsErrorCodeDescription := 'Device not initialized.';
    AdsErrorCodes.ADSERR_DEVICE_TIMEOUT:
        AdsErrorCodeDescription := 'Device has a timeout.';
    AdsErrorCodes.ADSERR_DEVICE_NOINTERFACE:
        AdsErrorCodeDescription := 'Interface query failed.';
    AdsErrorCodes.ADSERR_DEVICE_INVALIDINTERFACE:
        AdsErrorCodeDescription := 'Wrong interface requested.';
    AdsErrorCodes.ADSERR_DEVICE_INVALIDCLSID:
        AdsErrorCodeDescription := 'Class ID is invalid.';
    AdsErrorCodes.ADSERR_DEVICE_INVALIDOBJID:
        AdsErrorCodeDescription := 'Object ID is invalid.';
    AdsErrorCodes.ADSERR_DEVICE_PENDING:
        AdsErrorCodeDescription := 'Request pending.';
    AdsErrorCodes.ADSERR_DEVICE_ABORTED:
        AdsErrorCodeDescription := 'Request is aborted.';
    AdsErrorCodes.ADSERR_DEVICE_WARNING:
        AdsErrorCodeDescription := 'Signal warning.';
    AdsErrorCodes.ADSERR_DEVICE_INVALIDARRAYIDX:
        AdsErrorCodeDescription := 'Invalid array index.';
    AdsErrorCodes.ADSERR_DEVICE_SYMBOLNOTACTIVE:
        AdsErrorCodeDescription := 'Symbol not active.';
    AdsErrorCodes.ADSERR_DEVICE_ACCESSDENIED:
        AdsErrorCodeDescription := 'Access denied.';
    AdsErrorCodes.ADSERR_DEVICE_LICENSENOTFOUND:
        AdsErrorCodeDescription := 'Missing license.';
    AdsErrorCodes.ADSERR_DEVICE_LICENSEEXPIRED:
        AdsErrorCodeDescription := 'License expired.';
    AdsErrorCodes.ADSERR_DEVICE_LICENSEEXCEEDED:
        AdsErrorCodeDescription := 'License exceeded.';
    AdsErrorCodes.ADSERR_DEVICE_LICENSEINVALID:
        AdsErrorCodeDescription := 'Invalid license.';
    AdsErrorCodes.ADSERR_DEVICE_LICENSESYSTEMID:
        AdsErrorCodeDescription := 'License problem: System ID is invalid.';
    AdsErrorCodes.ADSERR_DEVICE_LICENSENOTIMELIMIT:
        AdsErrorCodeDescription := 'License not limited in time.';
    AdsErrorCodes.ADSERR_DEVICE_LICENSEFUTUREISSUE:
        AdsErrorCodeDescription := 'License problem: Time in the future.';
    AdsErrorCodes.ADSERR_DEVICE_LICENSETIMETOLONG:
        AdsErrorCodeDescription := 'License period too long.';
    AdsErrorCodes.ADSERR_DEVICE_EXCEPTION:
        AdsErrorCodeDescription := 'Exception at system startup.';
    AdsErrorCodes.ADSERR_DEVICE_LICENSEDUPLICATED:
        AdsErrorCodeDescription := 'License file read twice.';
    AdsErrorCodes.ADSERR_DEVICE_SIGNATUREINVALID:
        AdsErrorCodeDescription := 'Invalid signature.';
    AdsErrorCodes.ADSERR_DEVICE_CERTIFICATEINVALID:
        AdsErrorCodeDescription := 'Invalid certificate.';
    AdsErrorCodes.ADSERR_DEVICE_LICENSEOEMNOTFOUND:
        AdsErrorCodeDescription := 'Public key not known from OEM.';
    AdsErrorCodes.ADSERR_DEVICE_LICENSERESTRICTED:
        AdsErrorCodeDescription := 'License not valid for this system ID.';
    AdsErrorCodes.ADSERR_DEVICE_LICENSEDEMODENIED:
        AdsErrorCodeDescription := 'Demo license prohibited.';
    AdsErrorCodes.ADSERR_DEVICE_INVALIDFNCID:
        AdsErrorCodeDescription := 'Invalid function ID.';
    AdsErrorCodes.ADSERR_DEVICE_OUTOFRANGE:
        AdsErrorCodeDescription := 'Outside the valid range.';
    AdsErrorCodes.ADSERR_DEVICE_INVALIDALIGNMENT:
        AdsErrorCodeDescription := 'Invalid alignment.';
    AdsErrorCodes.ADSERR_DEVICE_LICENSEPLATFORM:
        AdsErrorCodeDescription := 'Invalid platform level.';
    AdsErrorCodes.ADSERR_DEVICE_FORWARD_PL:
        AdsErrorCodeDescription := 'Context – forward to passive level.';
    AdsErrorCodes.ADSERR_DEVICE_FORWARD_DL:
        AdsErrorCodeDescription := 'Context – forward to dispatch level.';
    AdsErrorCodes.ADSERR_DEVICE_FORWARD_RT:
        AdsErrorCodeDescription := 'Context – forward to real-time.';
    AdsErrorCodes.ADSERR_CLIENT_ERROR:
        AdsErrorCodeDescription := 'Client error.';
    AdsErrorCodes.ADSERR_CLIENT_INVALIDPARM:
        AdsErrorCodeDescription := 'Service contains an invalid parameter.';
    AdsErrorCodes.ADSERR_CLIENT_LISTEMPTY:
        AdsErrorCodeDescription := 'Polling list is empty.';
    AdsErrorCodes.ADSERR_CLIENT_VARUSED:
        AdsErrorCodeDescription := 'Var connection already in use.';
    AdsErrorCodes.ADSERR_CLIENT_DUPLINVOKEID:
        AdsErrorCodeDescription := 'The called ID is already in use.';
    AdsErrorCodes.ADSERR_CLIENT_SYNCTIMEOUT:
        AdsErrorCodeDescription := 'Timeout has occurred – the remote terminal is not responding in the specified ADS timeout. The route setting of the remote terminal may be configured incorrectly.';
    AdsErrorCodes.ADSERR_CLIENT_W32ERROR:
        AdsErrorCodeDescription := 'Error in Win32 subsystem.';
    AdsErrorCodes.ADSERR_CLIENT_TIMEOUTINVALID:
        AdsErrorCodeDescription := 'Invalid client timeout value.';
    AdsErrorCodes.ADSERR_CLIENT_PORTNOTOPEN:
        AdsErrorCodeDescription := 'Port not open.';
    AdsErrorCodes.ADSERR_CLIENT_NOAMSADDR:
        AdsErrorCodeDescription := 'No AMS address.';
    AdsErrorCodes.ADSERR_CLIENT_SYNCINTERNAL:
        AdsErrorCodeDescription := 'Internal error in Ads sync.';
    AdsErrorCodes.ADSERR_CLIENT_ADDHASH:
        AdsErrorCodeDescription := 'Hash table overflow.';
    AdsErrorCodes.ADSERR_CLIENT_REMOVEHASH:
        AdsErrorCodeDescription := 'Key not found in the table.';
    AdsErrorCodes.ADSERR_CLIENT_NOMORESYM:
        AdsErrorCodeDescription := 'No symbols in the cache.';
    AdsErrorCodes.ADSERR_CLIENT_SYNCRESINVALID:
        AdsErrorCodeDescription := 'Invalid response received.';
    AdsErrorCodes.ADSERR_CLIENT_SYNCPORTLOCKED:
        AdsErrorCodeDescription := 'Sync Port is locked.';
    AdsErrorCodes.RTERR_INTERNAL:
        AdsErrorCodeDescription := 'Internal error in the real-time system.';
    AdsErrorCodes.RTERR_BADTIMERPERIODS:
        AdsErrorCodeDescription := 'Timer value is not valid.';
    AdsErrorCodes.RTERR_INVALIDTASKPTR:
        AdsErrorCodeDescription := 'Task pointer has the invalid value 0 (zero).';
    AdsErrorCodes.RTERR_INVALIDSTACKPTR:
        AdsErrorCodeDescription := 'Stack pointer has the invalid value 0 (zero).';
    AdsErrorCodes.RTERR_PRIOEXISTS:
        AdsErrorCodeDescription := 'The request task priority is already assigned.';
    AdsErrorCodes.RTERR_NOMORETCB:
        AdsErrorCodeDescription :=
            'No free TCB (Task Control Block) available. The maximum number of TCBs is 64.';
    AdsErrorCodes.RTERR_NOMORESEMAS:
        AdsErrorCodeDescription :=
            'No free semaphores available. The maximum number of semaphores is 64.';
    AdsErrorCodes.RTERR_NOMOREQUEUES:
        AdsErrorCodeDescription :=
            'No free space available in the queue. The maximum number of positions in the queue is 64.';
    AdsErrorCodes.RTERR_EXTIRQALREADYDEF:
        AdsErrorCodeDescription := 'An external synchronization interrupt is already applied.';
    AdsErrorCodes.RTERR_EXTIRQNOTDEF:
        AdsErrorCodeDescription := 'No external sync interrupt applied.';
    AdsErrorCodes.RTERR_EXTIRQINSTALLFAILED:
        AdsErrorCodeDescription :=
            'Application of the external synchronization interrupt has failed.';
    AdsErrorCodes.RTERR_IRQLNOTLESSOREQUAL:
        AdsErrorCodeDescription := 'Call of a service function in the wrong context';
    AdsErrorCodes.RTERR_VMXNOTSUPPORTED:
        AdsErrorCodeDescription := 'Intel VT-x extension is not supported.';
    AdsErrorCodes.RTERR_VMXDISABLED:
        AdsErrorCodeDescription := 'Intel VT-x extension is not enabled in the BIOS.';
    AdsErrorCodes.RTERR_VMXCONTROLSMISSING:
        AdsErrorCodeDescription := 'Missing function in Intel VT-x extension.';
    AdsErrorCodes.RTERR_VMXENABLEFAILS:
        AdsErrorCodeDescription := 'Activation of Intel VT-x fails.';
    AdsErrorCodes.WSAETIMEDOUT:
        AdsErrorCodeDescription := 'A connection timeout has occurred while establishing the connection. Either the remote terminal did not respond properly after a certain period of time, or the established connection could not be maintained because the connected host did not respond.';
    AdsErrorCodes.WSAECONNREFUSED:
        AdsErrorCodeDescription := 'Connection refused. Connection couldnt be established because the target computer has rejected it. Error can result from an attempt to connect to a service that is inactive on the external host, i.e. a service for which no server application is running.';
    AdsErrorCodes.WSAEHOSTUNREACH:
        AdsErrorCodeDescription :=
            'No route to host - a socket operation referred to an unavailable host.';
ELSE
    AdsErrorCodeDescription := 'Unknown ADS error code.';
END_CASE

END_FUNCTION

// ---- ADS/ToAdsErrorCode.TcPOU
(*
Convert an ADS error code of type UDINT to the AdsErrorCodes datatype.

## Example
```
adsErrorId := 1802;
adsErrorCode := TcError.ToAdsErrorCode(adsErrorId); // ADSERR_DEVICE_NOMEMORY;
```

## Source
https://infosys.beckhoff.com/english.php?content=../content/1033/tf6701_tc3_iot_communication_mqtt/374277003.html&id=
*)
FUNCTION ToAdsErrorCode : AdsErrorCodes
VAR_INPUT
    errorCode : UDINT;
END_VAR

CASE errorCode OF
    0:
        ToAdsErrorCode := AdsErrorCodes.ERR_NOERROR;
    1:
        ToAdsErrorCode := AdsErrorCodes.ERR_INTERNAL;
    2:
        ToAdsErrorCode := AdsErrorCodes.ERR_NORTIME;
    3:
        ToAdsErrorCode := AdsErrorCodes.ERR_ALLOCLOCKEDMEM;
    4:
        ToAdsErrorCode := AdsErrorCodes.ERR_INSERTMAILBOX;
    5:
        ToAdsErrorCode := AdsErrorCodes.ERR_WRONGRECEIVEHMSG;
    6:
        ToAdsErrorCode := AdsErrorCodes.ERR_TARGETPORTNOTFOUND;
    7:
        ToAdsErrorCode := AdsErrorCodes.ERR_TARGETMACHINENOTFOUND;
    8:
        ToAdsErrorCode := AdsErrorCodes.ERR_UNKNOWNCMDID;
    9:
        ToAdsErrorCode := AdsErrorCodes.ERR_BADTASKID;
    10:
        ToAdsErrorCode := AdsErrorCodes.ERR_NOIO;
    11:
        ToAdsErrorCode := AdsErrorCodes.ERR_UNKNOWNAMSCMD;
    12:
        ToAdsErrorCode := AdsErrorCodes.ERR_WIN32ERROR;
    13:
        ToAdsErrorCode := AdsErrorCodes.ERR_PORTNOTCONNECTED;
    14:
        ToAdsErrorCode := AdsErrorCodes.ERR_INVALIDAMSLENGTH;
    15:
        ToAdsErrorCode := AdsErrorCodes.ERR_INVALIDAMSNETID;
    16:
        ToAdsErrorCode := AdsErrorCodes.ERR_LOWINSTLEVEL;
    17:
        ToAdsErrorCode := AdsErrorCodes.ERR_NODEBUGINTAVAILABLE;
    18:
        ToAdsErrorCode := AdsErrorCodes.ERR_PORTDISABLED;
    19:
        ToAdsErrorCode := AdsErrorCodes.ERR_PORTALREADYCONNECTED;
    20:
        ToAdsErrorCode := AdsErrorCodes.ERR_AMSSYNC_W32ERROR;
    21:
        ToAdsErrorCode := AdsErrorCodes.ERR_AMSSYNC_TIMEOUT;
    22:
        ToAdsErrorCode := AdsErrorCodes.ERR_AMSSYNC_AMSERROR;
    23:
        ToAdsErrorCode := AdsErrorCodes.ERR_AMSSYNC_NOINDEXINMAP;
    24:
        ToAdsErrorCode := AdsErrorCodes.ERR_INVALIDAMSPORT;
    25:
        ToAdsErrorCode := AdsErrorCodes.ERR_NOMEMORY;
    26:
        ToAdsErrorCode := AdsErrorCodes.ERR_TCPSEND;
    27:
        ToAdsErrorCode := AdsErrorCodes.ERR_HOSTUNREACHABLE;
    28:
        ToAdsErrorCode := AdsErrorCodes.ERR_INVALIDAMSFRAGMENT;
    29:
        ToAdsErrorCode := AdsErrorCodes.ERR_TLSSEND;
    30:
        ToAdsErrorCode := AdsErrorCodes.ERR_ACCESSDENIED;
    1280:
        ToAdsErrorCode := AdsErrorCodes.ROUTERERR_NOLOCKEDMEMORY;
    1281:
        ToAdsErrorCode := AdsErrorCodes.ROUTERERR_RESIZEMEMORY;
    1282:
        ToAdsErrorCode := AdsErrorCodes.ROUTERERR_MAILBOXFULL;
    1283:
        ToAdsErrorCode := AdsErrorCodes.ROUTERERR_DEBUGBOXFULL;
    1284:
        ToAdsErrorCode := AdsErrorCodes.ROUTERERR_UNKNOWNPORTTYPE;
    1285:
        ToAdsErrorCode := AdsErrorCodes.ROUTERERR_NOTINITIALIZED;
    1286:
        ToAdsErrorCode := AdsErrorCodes.ROUTERERR_PORTALREADYINUSE;
    1287:
        ToAdsErrorCode := AdsErrorCodes.ROUTERERR_NOTREGISTERED;
    1288:
        ToAdsErrorCode := AdsErrorCodes.ROUTERERR_NOMOREQUEUES;
    1289:
        ToAdsErrorCode := AdsErrorCodes.ROUTERERR_INVALIDPORT;
    1290:
        ToAdsErrorCode := AdsErrorCodes.ROUTERERR_NOTACTIVATED;
    1291:
        ToAdsErrorCode := AdsErrorCodes.ROUTERERR_FRAGMENTBOXFULL;
    1292:
        ToAdsErrorCode := AdsErrorCodes.ROUTERERR_FRAGMENTTIMEOUT;
    1293:
        ToAdsErrorCode := AdsErrorCodes.ROUTERERR_TOBEREMOVED;
    1792:
        ToAdsErrorCode := AdsErrorCodes.ADSERR_DEVICE_ERROR;
    1793:
        ToAdsErrorCode := AdsErrorCodes.ADSERR_DEVICE_SRVNOTSUPP;
    1794:
        ToAdsErrorCode := AdsErrorCodes.ADSERR_DEVICE_INVALIDGRP;
    1795:
        ToAdsErrorCode := AdsErrorCodes.ADSERR_DEVICE_INVALIDOFFSET;
    1796:
        ToAdsErrorCode := AdsErrorCodes.ADSERR_DEVICE_INVALIDACCESS;
    1797:
        ToAdsErrorCode := AdsErrorCodes.ADSERR_DEVICE_INVALIDSIZE;
    1798:
        ToAdsErrorCode := AdsErrorCodes.ADSERR_DEVICE_INVALIDDATA;
    1799:
        ToAdsErrorCode := AdsErrorCodes.ADSERR_DEVICE_NOTREADY;
    1800:
        ToAdsErrorCode := AdsErrorCodes.ADSERR_DEVICE_BUSY;
    1801:
        ToAdsErrorCode := AdsErrorCodes.ADSERR_DEVICE_INVALIDCONTEXT;
    1802:
        ToAdsErrorCode := AdsErrorCodes.ADSERR_DEVICE_NOMEMORY;
    1803:
        ToAdsErrorCode := AdsErrorCodes.ADSERR_DEVICE_INVALIDPARM;
    1804:
        ToAdsErrorCode := AdsErrorCodes.ADSERR_DEVICE_NOTFOUND;
    1805:
        ToAdsErrorCode := AdsErrorCodes.ADSERR_DEVICE_SYNTAX;
    1806:
        ToAdsErrorCode := AdsErrorCodes.ADSERR_DEVICE_INCOMPATIBLE;
    1807:
        ToAdsErrorCode := AdsErrorCodes.ADSERR_DEVICE_EXISTS;
    1808:
        ToAdsErrorCode := AdsErrorCodes.ADSERR_DEVICE_SYMBOLNOTFOUND;
    1809:
        ToAdsErrorCode := AdsErrorCodes.ADSERR_DEVICE_SYMBOLVERSIONINVALID;
    1810:
        ToAdsErrorCode := AdsErrorCodes.ADSERR_DEVICE_INVALIDSTATE;
    1811:
        ToAdsErrorCode := AdsErrorCodes.ADSERR_DEVICE_TRANSMODENOTSUPP;
    1812:
        ToAdsErrorCode := AdsErrorCodes.ADSERR_DEVICE_NOTIFYHNDINVALID;
    1813:
        ToAdsErrorCode := AdsErrorCodes.ADSERR_DEVICE_CLIENTUNKNOWN;
    1814:
        ToAdsErrorCode := AdsErrorCodes.ADSERR_DEVICE_NOMOREHDLS;
    1815:
        ToAdsErrorCode := AdsErrorCodes.ADSERR_DEVICE_INVALIDWATCHSIZE;
    1816:
        ToAdsErrorCode := AdsErrorCodes.ADSERR_DEVICE_NOTINIT;
    1817:
        ToAdsErrorCode := AdsErrorCodes.ADSERR_DEVICE_TIMEOUT;
    1818:
        ToAdsErrorCode := AdsErrorCodes.ADSERR_DEVICE_NOINTERFACE;
    1819:
        ToAdsErrorCode := AdsErrorCodes.ADSERR_DEVICE_INVALIDINTERFACE;
    1820:
        ToAdsErrorCode := AdsErrorCodes.ADSERR_DEVICE_INVALIDCLSID;
    1821:
        ToAdsErrorCode := AdsErrorCodes.ADSERR_DEVICE_INVALIDOBJID;
    1822:
        ToAdsErrorCode := AdsErrorCodes.ADSERR_DEVICE_PENDING;
    1823:
        ToAdsErrorCode := AdsErrorCodes.ADSERR_DEVICE_ABORTED;
    1824:
        ToAdsErrorCode := AdsErrorCodes.ADSERR_DEVICE_WARNING;
    1825:
        ToAdsErrorCode := AdsErrorCodes.ADSERR_DEVICE_INVALIDARRAYIDX;
    1826:
        ToAdsErrorCode := AdsErrorCodes.ADSERR_DEVICE_SYMBOLNOTACTIVE;
    1827:
        ToAdsErrorCode := AdsErrorCodes.ADSERR_DEVICE_ACCESSDENIED;
    1828:
        ToAdsErrorCode := AdsErrorCodes.ADSERR_DEVICE_LICENSENOTFOUND;
    1829:
        ToAdsErrorCode := AdsErrorCodes.ADSERR_DEVICE_LICENSEEXPIRED;
    1830:
        ToAdsErrorCode := AdsErrorCodes.ADSERR_DEVICE_LICENSEEXCEEDED;
    1831:
        ToAdsErrorCode := AdsErrorCodes.ADSERR_DEVICE_LICENSEINVALID;
    1832:
        ToAdsErrorCode := AdsErrorCodes.ADSERR_DEVICE_LICENSESYSTEMID;
    1833:
        ToAdsErrorCode := AdsErrorCodes.ADSERR_DEVICE_LICENSENOTIMELIMIT;
    1834:
        ToAdsErrorCode := AdsErrorCodes.ADSERR_DEVICE_LICENSEFUTUREISSUE;
    1835:
        ToAdsErrorCode := AdsErrorCodes.ADSERR_DEVICE_LICENSETIMETOLONG;
    1836:
        ToAdsErrorCode := AdsErrorCodes.ADSERR_DEVICE_EXCEPTION;
    1837:
        ToAdsErrorCode := AdsErrorCodes.ADSERR_DEVICE_LICENSEDUPLICATED;
    1838:
        ToAdsErrorCode := AdsErrorCodes.ADSERR_DEVICE_SIGNATUREINVALID;
    1839:
        ToAdsErrorCode := AdsErrorCodes.ADSERR_DEVICE_CERTIFICATEINVALID;
    1840:
        ToAdsErrorCode := AdsErrorCodes.ADSERR_DEVICE_LICENSEOEMNOTFOUND;
    1841:
        ToAdsErrorCode := AdsErrorCodes.ADSERR_DEVICE_LICENSERESTRICTED;
    1842:
        ToAdsErrorCode := AdsErrorCodes.ADSERR_DEVICE_LICENSEDEMODENIED;
    1843:
        ToAdsErrorCode := AdsErrorCodes.ADSERR_DEVICE_INVALIDFNCID;
    1844:
        ToAdsErrorCode := AdsErrorCodes.ADSERR_DEVICE_OUTOFRANGE;
    1845:
        ToAdsErrorCode := AdsErrorCodes.ADSERR_DEVICE_INVALIDALIGNMENT;
    1846:
        ToAdsErrorCode := AdsErrorCodes.ADSERR_DEVICE_LICENSEPLATFORM;
    1847:
        ToAdsErrorCode := AdsErrorCodes.ADSERR_DEVICE_FORWARD_PL;
    1848:
        ToAdsErrorCode := AdsErrorCodes.ADSERR_DEVICE_FORWARD_DL;
    1849:
        ToAdsErrorCode := AdsErrorCodes.ADSERR_DEVICE_FORWARD_RT;
    1856:
        ToAdsErrorCode := AdsErrorCodes.ADSERR_CLIENT_ERROR;
    1857:
        ToAdsErrorCode := AdsErrorCodes.ADSERR_CLIENT_INVALIDPARM;
    1858:
        ToAdsErrorCode := AdsErrorCodes.ADSERR_CLIENT_LISTEMPTY;
    1859:
        ToAdsErrorCode := AdsErrorCodes.ADSERR_CLIENT_VARUSED;
    1860:
        ToAdsErrorCode := AdsErrorCodes.ADSERR_CLIENT_DUPLINVOKEID;
    1861:
        ToAdsErrorCode := AdsErrorCodes.ADSERR_CLIENT_SYNCTIMEOUT;
    1862:
        ToAdsErrorCode := AdsErrorCodes.ADSERR_CLIENT_W32ERROR;
    1863:
        ToAdsErrorCode := AdsErrorCodes.ADSERR_CLIENT_TIMEOUTINVALID;
    1864:
        ToAdsErrorCode := AdsErrorCodes.ADSERR_CLIENT_PORTNOTOPEN;
    1865:
        ToAdsErrorCode := AdsErrorCodes.ADSERR_CLIENT_NOAMSADDR;
    1872:
        ToAdsErrorCode := AdsErrorCodes.ADSERR_CLIENT_SYNCINTERNAL;
    1873:
        ToAdsErrorCode := AdsErrorCodes.ADSERR_CLIENT_ADDHASH;
    1874:
        ToAdsErrorCode := AdsErrorCodes.ADSERR_CLIENT_REMOVEHASH;
    1875:
        ToAdsErrorCode := AdsErrorCodes.ADSERR_CLIENT_NOMORESYM;
    1876:
        ToAdsErrorCode := AdsErrorCodes.ADSERR_CLIENT_SYNCRESINVALID;
    1877:
        ToAdsErrorCode := AdsErrorCodes.ADSERR_CLIENT_SYNCPORTLOCKED;
    4096:
        ToAdsErrorCode := AdsErrorCodes.RTERR_INTERNAL;
    4097:
        ToAdsErrorCode := AdsErrorCodes.RTERR_BADTIMERPERIODS;
    4098:
        ToAdsErrorCode := AdsErrorCodes.RTERR_INVALIDTASKPTR;
    4099:
        ToAdsErrorCode := AdsErrorCodes.RTERR_INVALIDSTACKPTR;
    4100:
        ToAdsErrorCode := AdsErrorCodes.RTERR_PRIOEXISTS;
    4101:
        ToAdsErrorCode := AdsErrorCodes.RTERR_NOMORETCB;
    4102:
        ToAdsErrorCode := AdsErrorCodes.RTERR_NOMORESEMAS;
    4103:
        ToAdsErrorCode := AdsErrorCodes.RTERR_NOMOREQUEUES;
ELSE
    ToAdsErrorCode := AdsErrorCodes.ERR_UNKNOWN;
END_CASE

END_FUNCTION
